// TIA Portal V20 export
FUNCTION_BLOCK "MotorStarter"   // FB2, LAD
   VAR RETAIN
      IO { S7_SetPoint := 'True'} : "MotorIOSet";
   END_VAR
   VAR
      RisingEdgeFlags : Array[0..3] of Bool;
      NegitiveSignalEdge : Array[0..1] of Bool;
      HrTotaliserTimerReset : Bool;
      EnableUPSTimeMS : DInt;
      ShutdownTimeMS : DInt;
      FTTimeMS : DInt;
      FaultTripTimer { S7_SetPoint := 'True'} : TON_TIME;
      FTSTimer { S7_SetPoint := 'True'} : TON_TIME;
      EnableUpstreamTimer { S7_SetPoint := 'True'} : TON_TIME;
      InHandReqPreStart { S7_SetPoint := 'True'} : TON_TIME;
      ShutdownTimer { S7_SetPoint := 'True'} : TON_TIME;
      GeneralDelayTimer { S7_SetPoint := 'True'} : TON_TIME;
   END_VAR
   VAR RETAIN
      HrTotaliserTimer { S7_SetPoint := 'True'} : TONR_TIME;
   END_VAR
   VAR
      RecentStartSignal : TOF_TIME;
      PreStartMemory : Bool;
      HandNegEdge : Bool;
      HandPosEdge : Bool;
   END_VAR
   VAR_TEMP
      "Time" : Real;
   END_VAR
   VAR_TEMP   // added for the SCL form of the ladder/FBD networks
      _w1 : Bool;
      _w2 : Bool;
   END_VAR
BEGIN

REGION Network 1: DOL Motor Start / Stop
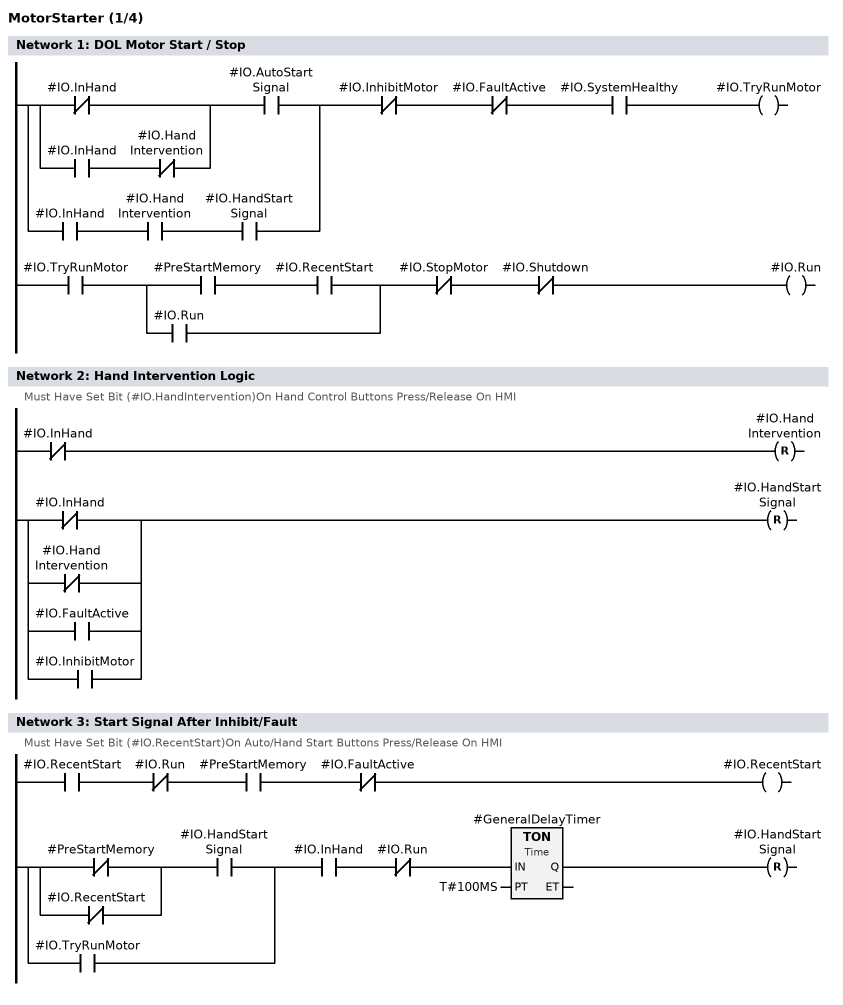
   RUNG wire#powerrail
      I_Contact( #IO.InHand )
      wire#w1
      Contact( #IO.AutoStartSignal )
      wire#w2
      I_Contact( #IO.InhibitMotor )
      I_Contact( #IO.FaultActive )
      Contact( #IO.SystemHealthy )
      Coil( #IO.TryRunMotor )
   END_RUNG
   RUNG wire#powerrail
      Contact( #IO.InHand )
      I_Contact( #IO.HandIntervention )
   END_RUNG wire#w1
   RUNG wire#powerrail
      Contact( #IO.InHand )
      Contact( #IO.HandIntervention )
      Contact( #IO.HandStartSignal )
   END_RUNG wire#w2
   RUNG wire#powerrail
      Contact( #IO.TryRunMotor )
      wire#w3
      Contact( #PreStartMemory )
      Contact( #IO.RecentStart )
      wire#w4
      I_Contact( #IO.StopMotor )
      I_Contact( #IO.Shutdown )
      Coil( #IO.Run )
   END_RUNG
   RUNG wire#w3
      Contact( #IO.Run )
   END_RUNG wire#w4
   // the same network as SCL:
   #IO.TryRunMotor := (((NOT #IO.InHand OR (#IO.InHand AND NOT #IO.HandIntervention)) AND #IO.AutoStartSignal) OR (#IO.InHand AND #IO.HandIntervention AND #IO.HandStartSignal)) AND NOT #IO.InhibitMotor AND NOT #IO.FaultActive AND #IO.SystemHealthy;
   #IO.Run := #IO.TryRunMotor AND ((#PreStartMemory AND #IO.RecentStart) OR #IO.Run) AND NOT #IO.StopMotor AND NOT #IO.Shutdown;
END_REGION

REGION Network 2: Hand Intervention Logic
   // Must Have Set Bit (#IO.HandIntervention)On Hand Control Buttons Press/Release On HMI
   RUNG wire#powerrail
      I_Contact( #IO.InHand )
      R_Coil( #IO.HandIntervention )
   END_RUNG
   RUNG wire#powerrail
      I_Contact( #IO.InHand )
      wire#w1
      R_Coil( #IO.HandStartSignal )
   END_RUNG
   RUNG wire#powerrail
      I_Contact( #IO.HandIntervention )
   END_RUNG wire#w1
   RUNG wire#powerrail
      Contact( #IO.FaultActive )
   END_RUNG wire#w1
   RUNG wire#powerrail
      Contact( #IO.InhibitMotor )
   END_RUNG wire#w1
   // the same network as SCL:
   IF NOT #IO.InHand THEN #IO.HandIntervention := FALSE; END_IF;
   IF NOT #IO.InHand OR NOT #IO.HandIntervention OR #IO.FaultActive OR #IO.InhibitMotor THEN
       #IO.HandStartSignal := FALSE;
   END_IF;
END_REGION

REGION Network 3: Start Signal After Inhibit/Fault
   // Must Have Set Bit (#IO.RecentStart)On Auto/Hand Start Buttons Press/Release On HMI
   RUNG wire#powerrail
      Contact( #IO.RecentStart )
      I_Contact( #IO.Run )
      Contact( #PreStartMemory )
      I_Contact( #IO.FaultActive )
      Coil( #IO.RecentStart )
   END_RUNG
   RUNG wire#powerrail
      I_Contact( #PreStartMemory )
      wire#w1
      Contact( #IO.HandStartSignal )
      wire#w2
      Contact( #IO.InHand )
      I_Contact( #IO.Run )
      { S7_Templates := "time_type := Time" } #GeneralDelayTimer.TON(pt := T#100MS, et =>)
      R_Coil( #IO.HandStartSignal )
   END_RUNG
   RUNG wire#powerrail
      I_Contact( #IO.RecentStart )
   END_RUNG wire#w1
   RUNG wire#powerrail
      Contact( #IO.TryRunMotor )
   END_RUNG wire#w2
   // the same network as SCL:
   #IO.RecentStart := #IO.RecentStart AND NOT #IO.Run AND #PreStartMemory AND NOT #IO.FaultActive;
   #GeneralDelayTimer(IN := (((NOT #PreStartMemory OR NOT #IO.RecentStart) AND #IO.HandStartSignal) OR #IO.TryRunMotor) AND #IO.InHand AND NOT #IO.Run,   // TON
                      PT := T#100MS);
   IF #GeneralDelayTimer.Q THEN #IO.HandStartSignal := FALSE; END_IF;
END_REGION

REGION Network 4
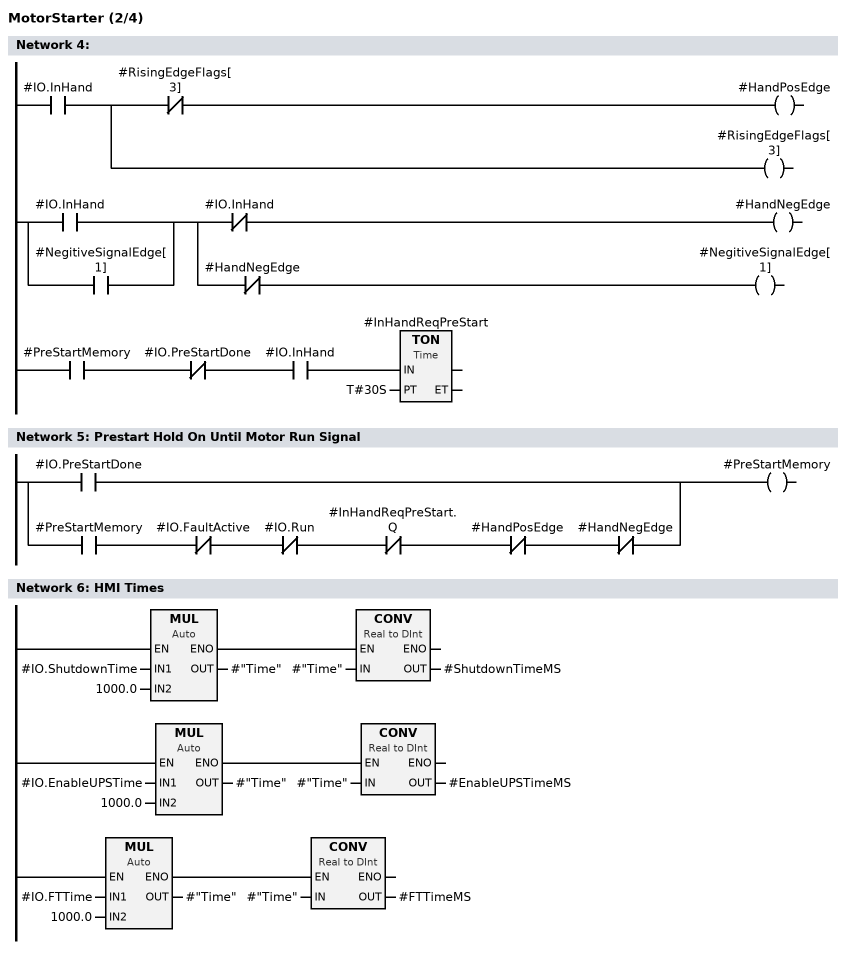
   RUNG wire#powerrail
      Contact( #IO.InHand )
      wire#w1
      I_Contact( #RisingEdgeFlags[3] )
      Coil( #HandPosEdge )
   END_RUNG
   RUNG wire#w1
      Coil( #RisingEdgeFlags[3] )
   END_RUNG
   RUNG wire#powerrail
      Contact( #IO.InHand )
      wire#w2
      I_Contact( #IO.InHand )
      Coil( #HandNegEdge )
   END_RUNG
   RUNG wire#powerrail
      Contact( #NegitiveSignalEdge[1] )
   END_RUNG wire#w2
   RUNG wire#w2
      I_Contact( #HandNegEdge )
      Coil( #NegitiveSignalEdge[1] )
   END_RUNG
   RUNG wire#powerrail
      Contact( #PreStartMemory )
      I_Contact( #IO.PreStartDone )
      Contact( #IO.InHand )
      { S7_Templates := "time_type := Time" } #InHandReqPreStart.TON(pt := T#30S, et =>)
   END_RUNG
   // the same network as SCL:
   #HandPosEdge := #IO.InHand AND NOT #RisingEdgeFlags[3];
   #RisingEdgeFlags[3] := #IO.InHand;
   #_w1 := #IO.InHand OR #NegitiveSignalEdge[1];
   #HandNegEdge := #_w1 AND NOT #IO.InHand;
   #NegitiveSignalEdge[1] := #_w1 AND NOT #HandNegEdge;
   #InHandReqPreStart(IN := #PreStartMemory AND NOT #IO.PreStartDone AND #IO.InHand, PT := T#30S);   // TON
END_REGION

REGION Network 5: Prestart Hold On Until Motor Run Signal
   RUNG wire#powerrail
      Contact( #IO.PreStartDone )
      wire#w1
      Coil( #PreStartMemory )
   END_RUNG
   RUNG wire#powerrail
      Contact( #PreStartMemory )
      I_Contact( #IO.FaultActive )
      I_Contact( #IO.Run )
      I_Contact( #InHandReqPreStart.Q )
      I_Contact( #HandPosEdge )
      I_Contact( #HandNegEdge )
   END_RUNG wire#w1
   // the same network as SCL:
   #PreStartMemory := #IO.PreStartDone OR (#PreStartMemory AND NOT #IO.FaultActive AND NOT #IO.Run AND NOT #InHandReqPreStart.Q AND NOT #HandPosEdge AND NOT #HandNegEdge);
END_REGION

REGION Network 6: HMI Times
   RUNG wire#powerrail
      Mul(in1 := #IO.ShutdownTime, in2 := 1000.0, out => #"Time")
      { S7_Templates := "[SrcType := Real, DestType := DInt]" } Convert(in := #"Time", out => #ShutdownTimeMS)
   END_RUNG
   RUNG wire#powerrail
      Mul(in1 := #IO.EnableUPSTime, in2 := 1000.0, out => #"Time")
      { S7_Templates := "[SrcType := Real, DestType := DInt]" } Convert(in := #"Time", out => #EnableUPSTimeMS)
   END_RUNG
   RUNG wire#powerrail
      Mul(in1 := #IO.FTTime, in2 := 1000.0, out => #"Time")
      { S7_Templates := "[SrcType := Real, DestType := DInt]" } Convert(in := #"Time", out => #FTTimeMS)
   END_RUNG
   // the same network as SCL:
   #"Time" := #IO.ShutdownTime * 1000.0;
   #ShutdownTimeMS := REAL_TO_DINT(#"Time");
   #"Time" := #IO.EnableUPSTime * 1000.0;
   #EnableUPSTimeMS := REAL_TO_DINT(#"Time");
   #"Time" := #IO.FTTime * 1000.0;
   #FTTimeMS := REAL_TO_DINT(#"Time");
END_REGION

REGION Network 7: DOL Motor Shutdown
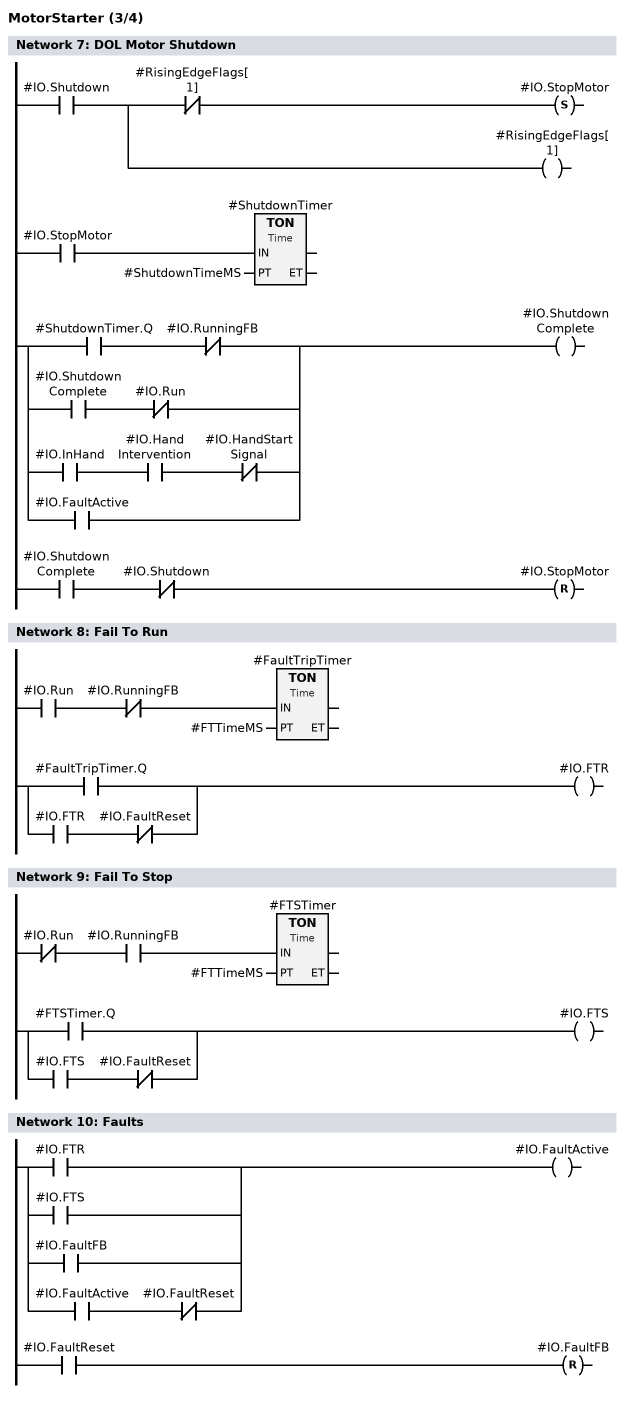
   RUNG wire#powerrail
      Contact( #IO.Shutdown )
      wire#w1
      I_Contact( #RisingEdgeFlags[1] )
      S_Coil( #IO.StopMotor )
   END_RUNG
   RUNG wire#w1
      Coil( #RisingEdgeFlags[1] )
   END_RUNG
   RUNG wire#powerrail
      Contact( #IO.StopMotor )
      { S7_Templates := "time_type := Time" } #ShutdownTimer.TON(pt := #ShutdownTimeMS, et =>)
   END_RUNG
   RUNG wire#powerrail
      Contact( #ShutdownTimer.Q )
      I_Contact( #IO.RunningFB )
      wire#w2
      Coil( #IO.ShutdownComplete )
   END_RUNG
   RUNG wire#powerrail
      Contact( #IO.ShutdownComplete )
      I_Contact( #IO.Run )
   END_RUNG wire#w2
   RUNG wire#powerrail
      Contact( #IO.InHand )
      Contact( #IO.HandIntervention )
      I_Contact( #IO.HandStartSignal )
   END_RUNG wire#w2
   RUNG wire#powerrail
      Contact( #IO.FaultActive )
   END_RUNG wire#w2
   RUNG wire#powerrail
      Contact( #IO.ShutdownComplete )
      I_Contact( #IO.Shutdown )
      R_Coil( #IO.StopMotor )
   END_RUNG
   // the same network as SCL:
   IF #IO.Shutdown AND NOT #RisingEdgeFlags[1] THEN #IO.StopMotor := TRUE; END_IF;
   #RisingEdgeFlags[1] := #IO.Shutdown;
   #ShutdownTimer(IN := #IO.StopMotor, PT := #ShutdownTimeMS);   // TON
   #IO.ShutdownComplete := (#ShutdownTimer.Q AND NOT #IO.RunningFB) OR (#IO.ShutdownComplete AND NOT #IO.Run) OR (#IO.InHand AND #IO.HandIntervention AND NOT #IO.HandStartSignal) OR #IO.FaultActive;
   IF #IO.ShutdownComplete AND NOT #IO.Shutdown THEN #IO.StopMotor := FALSE; END_IF;
END_REGION

REGION Network 8: Fail To Run
   RUNG wire#powerrail
      Contact( #IO.Run )
      I_Contact( #IO.RunningFB )
      { S7_Templates := "time_type := Time" } #FaultTripTimer.TON(pt := #FTTimeMS, et =>)
   END_RUNG
   RUNG wire#powerrail
      Contact( #FaultTripTimer.Q )
      wire#w1
      Coil( #IO.FTR )
   END_RUNG
   RUNG wire#powerrail
      Contact( #IO.FTR )
      I_Contact( #IO.FaultReset )
   END_RUNG wire#w1
   // the same network as SCL:
   #FaultTripTimer(IN := #IO.Run AND NOT #IO.RunningFB, PT := #FTTimeMS);   // TON
   #IO.FTR := #FaultTripTimer.Q OR (#IO.FTR AND NOT #IO.FaultReset);
END_REGION

REGION Network 9: Fail To Stop
   RUNG wire#powerrail
      I_Contact( #IO.Run )
      Contact( #IO.RunningFB )
      { S7_Templates := "time_type := Time" } #FTSTimer.TON(pt := #FTTimeMS, et =>)
   END_RUNG
   RUNG wire#powerrail
      Contact( #FTSTimer.Q )
      wire#w1
      Coil( #IO.FTS )
   END_RUNG
   RUNG wire#powerrail
      Contact( #IO.FTS )
      I_Contact( #IO.FaultReset )
   END_RUNG wire#w1
   // the same network as SCL:
   #FTSTimer(IN := NOT #IO.Run AND #IO.RunningFB, PT := #FTTimeMS);   // TON
   #IO.FTS := #FTSTimer.Q OR (#IO.FTS AND NOT #IO.FaultReset);
END_REGION

REGION Network 10: Faults
   RUNG wire#powerrail
      Contact( #IO.FTR )
      wire#w1
      Coil( #IO.FaultActive )
   END_RUNG
   RUNG wire#powerrail
      Contact( #IO.FTS )
   END_RUNG wire#w1
   RUNG wire#powerrail
      Contact( #IO.FaultFB )
   END_RUNG wire#w1
   RUNG wire#powerrail
      Contact( #IO.FaultActive )
      I_Contact( #IO.FaultReset )
   END_RUNG wire#w1
   RUNG wire#powerrail
      Contact( #IO.FaultReset )
      R_Coil( #IO.FaultFB )
   END_RUNG
   // the same network as SCL:
   #IO.FaultActive := #IO.FTR OR #IO.FTS OR #IO.FaultFB OR (#IO.FaultActive AND NOT #IO.FaultReset);
   IF #IO.FaultReset THEN #IO.FaultFB := FALSE; END_IF;
END_REGION

REGION Network 11: Motor Running, Enable Upstream Component
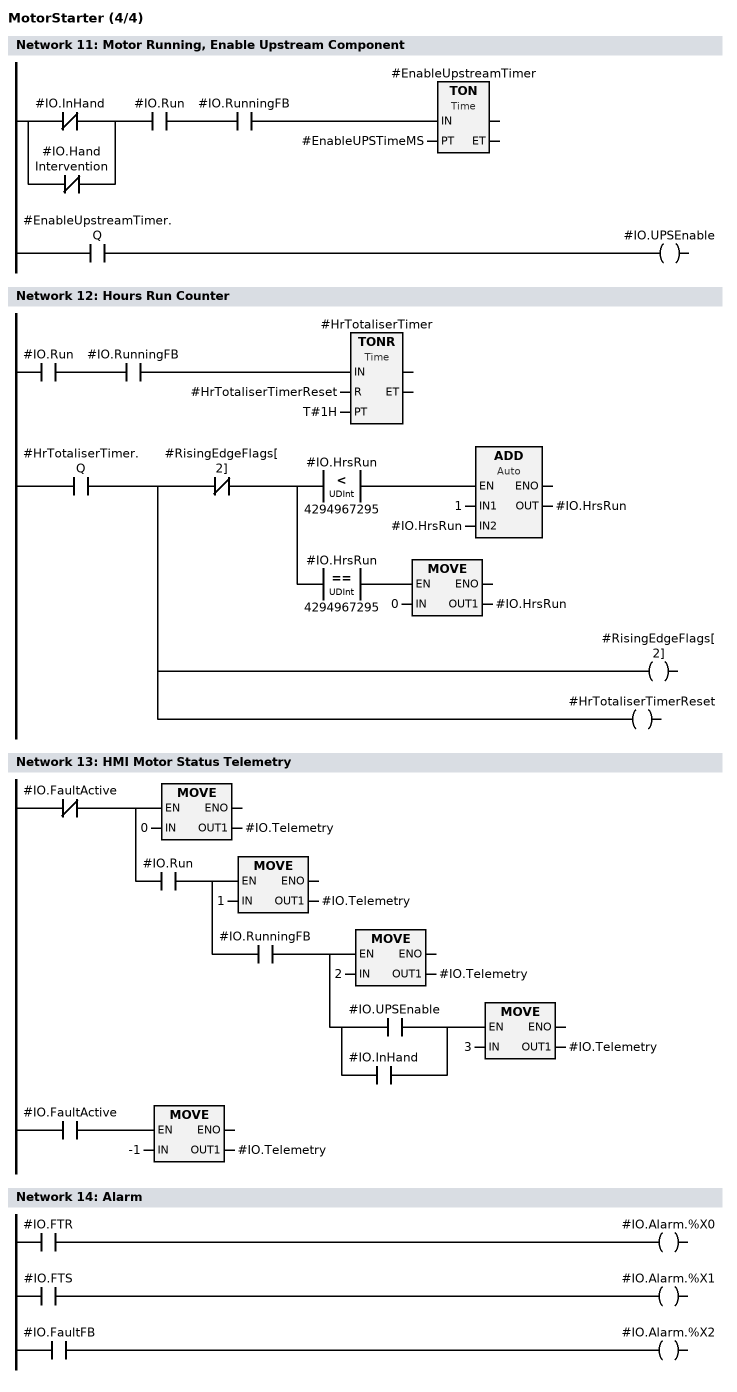
   RUNG wire#powerrail
      I_Contact( #IO.InHand )
      wire#w1
      Contact( #IO.Run )
      Contact( #IO.RunningFB )
      { S7_Templates := "time_type := Time" } #EnableUpstreamTimer.TON(pt := #EnableUPSTimeMS, et =>)
   END_RUNG
   RUNG wire#powerrail
      I_Contact( #IO.HandIntervention )
   END_RUNG wire#w1
   RUNG wire#powerrail
      Contact( #EnableUpstreamTimer.Q )
      Coil( #IO.UPSEnable )
   END_RUNG
   // the same network as SCL:
   #EnableUpstreamTimer(IN := (NOT #IO.InHand OR NOT #IO.HandIntervention) AND #IO.Run AND #IO.RunningFB,   // TON
                        PT := #EnableUPSTimeMS);
   #IO.UPSEnable := #EnableUpstreamTimer.Q;
END_REGION

REGION Network 12: Hours Run Counter
   RUNG wire#powerrail
      Contact( #IO.Run )
      Contact( #IO.RunningFB )
      { S7_Templates := "time_type := Time" } #HrTotaliserTimer.TONR(r := #HrTotaliserTimerReset, pt := T#1H, et =>)
   END_RUNG
   RUNG wire#powerrail
      Contact( #HrTotaliserTimer.Q )
      wire#w1
      I_Contact( #RisingEdgeFlags[2] )
      wire#w2
      { S7_Templates := "SrcType := UDInt" } LT_Contact(in1 := #IO.HrsRun, in2 := 4294967295)
      Add(in1 := 1, in2 := #IO.HrsRun, out => #IO.HrsRun)
   END_RUNG
   RUNG wire#w2
      { S7_Templates := "SrcType := UDInt" } EQ_Contact(in1 := #IO.HrsRun, in2 := 4294967295)
      Move(in := 0, out1 => #IO.HrsRun)
   END_RUNG
   RUNG wire#w1
      Coil( #RisingEdgeFlags[2] )
   END_RUNG
   RUNG wire#w1
      Coil( #HrTotaliserTimerReset )
   END_RUNG
   // the same network as SCL:
   #HrTotaliserTimer(IN := #IO.Run AND #IO.RunningFB, R := #HrTotaliserTimerReset, PT := T#1H);   // TONR
   #_w1 := #HrTotaliserTimer.Q AND NOT #RisingEdgeFlags[2];
   IF #_w1 AND (#IO.HrsRun < 4294967295) THEN #IO.HrsRun := 1 + #IO.HrsRun; END_IF;
   IF #_w1 AND (#IO.HrsRun = 4294967295) THEN #IO.HrsRun := 0; END_IF;
   #RisingEdgeFlags[2] := #HrTotaliserTimer.Q;
   #HrTotaliserTimerReset := #HrTotaliserTimer.Q;
END_REGION

REGION Network 13: HMI Motor Status Telemetry
   RUNG wire#powerrail
      I_Contact( #IO.FaultActive )
      wire#w1
      Move(in := 0, out1 => #IO.Telemetry)
   END_RUNG
   RUNG wire#w1
      Contact( #IO.Run )
      wire#w2
      Move(in := 1, out1 => #IO.Telemetry)
   END_RUNG
   RUNG wire#w2
      Contact( #IO.RunningFB )
      wire#w3
      Move(in := 2, out1 => #IO.Telemetry)
   END_RUNG
   RUNG wire#w3
      Contact( #IO.UPSEnable )
      wire#w4
      Move(in := 3, out1 => #IO.Telemetry)
   END_RUNG
   RUNG wire#w3
      Contact( #IO.InHand )
   END_RUNG wire#w4
   RUNG wire#powerrail
      Contact( #IO.FaultActive )
      Move(in := -1, out1 => #IO.Telemetry)
   END_RUNG
   // the same network as SCL:
   IF NOT #IO.FaultActive THEN #IO.Telemetry := 0; END_IF;
   #_w1 := NOT #IO.FaultActive AND #IO.Run;
   IF #_w1 THEN #IO.Telemetry := 1; END_IF;
   #_w2 := #_w1 AND #IO.RunningFB;
   IF #_w2 THEN #IO.Telemetry := 2; END_IF;
   IF #_w2 AND (#IO.UPSEnable OR #IO.InHand) THEN #IO.Telemetry := 3; END_IF;
   IF #IO.FaultActive THEN #IO.Telemetry := -1; END_IF;
END_REGION

REGION Network 14: Alarm
   RUNG wire#powerrail
      Contact( #IO.FTR )
      Coil( #IO.Alarm.%X0 )
   END_RUNG
   RUNG wire#powerrail
      Contact( #IO.FTS )
      Coil( #IO.Alarm.%X1 )
   END_RUNG
   RUNG wire#powerrail
      Contact( #IO.FaultFB )
      Coil( #IO.Alarm.%X2 )
   END_RUNG
   // the same network as SCL:
   #IO.Alarm.%X0 := #IO.FTR;
   #IO.Alarm.%X1 := #IO.FTS;
   #IO.Alarm.%X2 := #IO.FaultFB;
END_REGION
END_FUNCTION_BLOCK
